{attribute 'TcGenerated'}
// This function has been automatically generated from the project information.
VAR_GLOBAL CONSTANT
	{attribute 'const_non_replaced'}
	{attribute 'linkalways'}
	stLibVersion_tclib_ph_lv1_io : ST_LibVersion := (iMajor := 0, iMinor := 1, iBuild := 1, iRevision := 0, sVersion := '0.1.1.0');
END_VAR

(* stored: Version 1.1.0.1, ProductVersion 3.1.4019.2
   GVL Global_Version: Id {563c9f1a-97fd-402d-b145-afeac7f84f05} *)
